// TIA Portal V16 export
// export: Created 2021-11-12T13:32:31.3692651Z, ExportSetting WithDefaults, DisplayName Totally Integrated Automation Portal, DisplayVersion V16 Update 3, DisplayName TIA Portal Version Control Interface, DisplayVersion V16 Update 2, DisplayName TIA Portal Openness, DisplayVersion V16 Update 3, DisplayName SINAMICS Startdrive Advanced, DisplayVersion V16 Update 5, DisplayName SINAMICS Startdrive G130, G150, S120, S150, SINAMICS MV, S210, DisplayVersion V16 Update 5, DisplayName SINAMICS Startdrive G110M, G120, G120C, G120D, G120P, G115D, DisplayVersion V16 Update 5, DisplayName STEP 7 Professional, DisplayVersion V16 Update 3, DisplayName STEP 7 Safety, DisplayVersion V16, DisplayName WinCC UA Professional, DisplayVersion V16 Update 3
DATA_BLOCK "IDB_Station1R4"   // DB165
VERSION : 0.1
// stored: AutoNumber true, DBAccessibleFromOPCUA true, InstanceOfName Station1R4, InstanceOfType FB
"Station1R4"
   // VAR
   //    SF_RO01_Timeout : "STD_DI_Mon";
   //    SF_RO01_Lubrication : "STD_DI_Mon";
   //    SF_RC01 : "STD_DriveRobotABB";
   //    SF_RO01 : "STD_RobotABB";
   //    SF_RobotGripper : "STD_RobotGripper";
   //    SF_Sequence { S7_SetPoint := 'True'} : "Station 1R4 Seq";
   //    SF_Lubrication { S7_SetPoint := 'True'} : "TrackLubrication";
   //    SF_RobNotUsed { S7_SetPoint := 'True'} : "STD_OnOff";
   //    SS_RobotZones { S7_SetPoint := 'True'} : "STD_RobotZones";
   //    SS_Edge { S7_SetPoint := 'True'} : Array[0..100] of Bool;
   //    SDIPartId : DInt;
   //    SI_PartType : Int;
   //    SI_140RowNo { ExternalAccessible := 'False'; ExternalVisible := 'False'; ExternalWritable := 'False'} : Int;
   //    SI_140LineNo { ExternalAccessible := 'False'; ExternalVisible := 'False'; ExternalWritable := 'False'} : Int;
   //    SI_160RowNo { ExternalAccessible := 'False'; ExternalVisible := 'False'; ExternalWritable := 'False'} : Int;
   //    SI_160LineNo { ExternalAccessible := 'False'; ExternalVisible := 'False'; ExternalWritable := 'False'} : Int;
   //    SI_180RowNo { ExternalAccessible := 'False'; ExternalVisible := 'False'; ExternalWritable := 'False'} : Int;
   //    SI_180LineNo { ExternalAccessible := 'False'; ExternalVisible := 'False'; ExternalWritable := 'False'} : Int;
   //    SB1TakePosFound140 { ExternalAccessible := 'False'; ExternalVisible := 'False'; ExternalWritable := 'False'} : Bool;
   //    SB1PutPosFound160 { ExternalAccessible := 'False'; ExternalVisible := 'False'; ExternalWritable := 'False'} : Bool;
   //    SB1PutPosFound180 { ExternalAccessible := 'False'; ExternalVisible := 'False'; ExternalWritable := 'False'} : Bool;
   //    SB1ReqToChangeTool : Bool;
   //    SB1ChangeToolDone : Bool;
   //    SB1CycleAutostop : Bool;
   //    SB1ServicePosReq { ExternalAccessible := 'False'; ExternalVisible := 'False'; ExternalWritable := 'False'} : Bool;
   //    SB1LubricError : Bool;
   // END_VAR
BEGIN
END_DATA_BLOCK
